Staubli VAL3: recvRosMsg.pgx

public program recvRosMsg(RobotStatus& x_rRobotStatus, FlagStatus& x_fRosStatus, num x_nRosFlagCmd)
begin

  //This program is used for receiving motion planning command from the Host ROS controller and
  //ensuring the received ros massages correct.

  while true
    //Call the receive data function
    call recvData(siTcpIpMotion,nRecvData,x_rRobotStatus,x_fRosStatus,x_nRosFlagCmd)

    //Froce an end to the current task and enter the next sequence loop
    delay(0.0)

  endWhile

end
